PROGRAM INTERNAL PRG_TEST_FB_LOGTODISK
VAR
	fbLogToDisk : FB_LogToDisk(
						sLogFolder := '/tmp',
						sLogFilePrefix := 'AutomaticTestLog_',
						sLogFileExtension := 'txt',
						nMaxLogFileSize := 500,
						nMaxNumberOfLogFiles := 3
					);
	bEnableTests : BOOL;
	bEnable : BOOL;
	bAddToLog : BOOL;
	bStressTest : BOOL;
	nIdx : UDINT;
	sMsg : T_MaxString;
END_VAR

IF bEnableTests THEN
	fbLogToDisk(bEnable := bEnable);
	IF bAddToLog THEN
		bAddToLog := FALSE;
		fbLogToDisk.DEBUG(sMsg);
	END_IF
	IF bStressTest THEN
		// Write an item to the log every PLC cycle, this should trigger a buffer overflow
		nIdx := nIdx + 1;
		sMsg := UDINT_TO_STRING(nIdx);
		fbLogToDisk.DEBUG(sMsg);
	END_IF
END_IF

END_PROGRAM

(* stored: Version 1.1.0.1, ProductVersion 3.1.4024.11
   POU PRG_TEST_FB_LOGTODISK: Id {90bc222e-4655-0939-07a6-64349ec214b9}, SpecialFunc None *)
